{attribute 'linkalways'} 
{attribute 'no_explicit_call' := 'This FB is a CLASS and must be accessed using methods or properties'}
{attribute 'enable_dynamic_creation'}
FUNCTION_BLOCK PromiseContext IMPLEMENTS I_PromiseContext
VAR
	state : (PROMISE_PENDING, PROMISE_REJECTED, PROMISE_RESOLVED);
	reason : T_MAXSTRING;
	entities : Dictionary;
	pBuffer : POINTER TO BYTE;
	bufferSize : UDINT;
END_VAR

METHOD PRIVATE CopyBufferToDestination
VAR_INPUT
	DestinationAddress : PVOID;
END_VAR
MEMCPY(DestinationAddress, pBuffer, bufferSize);
END_METHOD

METHOD PRIVATE CopySourceToBuffer
VAR_INPUT
	SourceAddress : PVOID;
END_VAR
MEMCPY(pBuffer, SourceAddress, bufferSize);
END_METHOD

METHOD PRIVATE CreateBuffer
VAR_INPUT
	SizeInBytes : UDINT;
END_VAR
bufferSize := SizeInBytes;
pBuffer := __NEW(BYTE, SizeInBytes);
END_METHOD

METHOD PRIVATE DestroyBuffer
VAR_INPUT
END_VAR
IF pBuffer = 0 THEN
	RETURN;
END_IF

__DELETE(pBuffer);
bufferSize := 0;
END_METHOD

METHOD FB_exit : BOOL
VAR_INPUT
	bInCopyCode : BOOL; // if TRUE, the exit method is called for exiting an instance that is copied afterwards (online change).
END_VAR
IF bInCopyCode THEN
	RETURN;
END_IF

DestroyBuffer();
END_METHOD

PROPERTY PUBLIC Pending : BOOL
GET
Pending := state = PROMISE_PENDING;
END_GET
END_PROPERTY

METHOD PUBLIC Reject
VAR_INPUT
	Reason : T_MAXSTRING;
END_VAR
IF NOT Pending THEN
	RETURN;
END_IF

THIS^.reason := Reason;
state := PROMISE_REJECTED;
END_METHOD

PROPERTY Rejected : BOOL
GET
Rejected := state = PROMISE_REJECTED;
END_GET
END_PROPERTY

PROPERTY RejectedReason : T_MAXSTRING
GET
RejectedReason := reason;
END_GET
END_PROPERTY

METHOD PUBLIC Resolve
VAR_INPUT
END_VAR
IF NOT Pending THEN
	RETURN;
END_IF

state := PROMISE_RESOLVED;
END_METHOD

PROPERTY Resolved : BOOL
GET
Resolved := state = PROMISE_RESOLVED;
END_GET
END_PROPERTY

METHOD PUBLIC ResolveWith
VAR_INPUT
	Value : ANY;
END_VAR
IF NOT Pending THEN
	RETURN;
END_IF

state := PROMISE_RESOLVED;
CreateBuffer(DINT_TO_UDINT(Value.diSize));
CopySourceToBuffer(Value.pValue);
END_METHOD

METHOD PUBLIC TryGetEntity : BOOL
VAR_INPUT
	Key : T_MAXSTRING;
	Destination	: ANY;
END_VAR
TryGetEntity := entities.TryGetValue(Key, Destination);
END_METHOD

METHOD PUBLIC TryGetEntityTo : BOOL
VAR_INPUT
	Key : T_MAXSTRING;
	DestinationAddress : PVOID;
	DestinationSize : UDINT;
END_VAR
TryGetEntityTo := entities.TryGetValueTo(Key, DestinationAddress, DestinationSize);
END_METHOD

METHOD PUBLIC TryGetResult : BOOL
VAR_INPUT
	Destination : ANY;
END_VAR
IF NOT Resolved THEN
	RETURN;
END_IF

TryGetResult := TryGetResultTo(Destination.pValue, DINT_TO_UDINT(Destination.diSize));
END_METHOD

METHOD PUBLIC TryGetResultTo : BOOL
VAR_INPUT
	DestinationAddress : PVOID;
	DestinationSize : UDINT;
END_VAR
IF NOT Resolved THEN
	RETURN;
END_IF

IF pBuffer = 0 THEN
	RETURN;
END_IF

IF bufferSize <> DestinationSize THEN
	RETURN;
END_IF

CopyBufferToDestination(DestinationAddress);
TryGetResultTo := TRUE;
END_METHOD

METHOD PUBLIC TrySetEntity : BOOL
VAR_INPUT
	Key : T_MAXSTRING;
	Value : ANY;
END_VAR
TrySetEntity := entities.TryAdd(Key, Value);
END_METHOD

END_FUNCTION_BLOCK

(* stored: Version 1.1.0.1, ProductVersion 3.1.4024.12
   POU PromiseContext: Id {75de2a15-307e-435d-83d9-7a9c6fc0aa6b}, SpecialFunc None
   Folder Destructor: Id {3206c6d1-73ba-4bcb-9573-ef49dfe35813}
   Folder Private: Id {2aeb644b-aaad-4298-8cfb-e5854fe0a558}
   Method CopyBufferToDestination: Id {643053a8-761b-44b6-b0e6-941cdfc54020}
   Method CopySourceToBuffer: Id {18d0ddd0-a56f-44a7-8313-4f7aac18c40f}
   Method CreateBuffer: Id {d1c0e31e-bcae-46c4-a6b3-a9a2c7832b79}
   Method DestroyBuffer: Id {18a4e6b2-a240-42cc-907a-6394e5a913fc}
   Method FB_exit: Id {ed9e31bb-5056-4c6e-aecd-e284355dc15c}
   Property Pending: Id {3e6c5105-de16-4dc6-9419-c281f6072c9e}
   Get Get: Id {c8bcd943-4822-4043-8555-5d3c366f5060}
   Method Reject: Id {3005d554-6d2b-4118-bbde-742e87e3e26b}
   Property Rejected: Id {19b6e227-f6bc-4e54-bb57-3ef321fea3ee}
   Get Get: Id {a2e9ead9-bf2b-4df8-85d9-9300605aee90}
   Property RejectedReason: Id {54ee7955-fd3c-48fe-8732-72512e9a1ff9}
   Get Get: Id {f4b08042-2a5e-4864-8192-66c3e2b97f00}
   Method Resolve: Id {a6b23446-da8d-43df-9791-1e09c13c9a89}
   Property Resolved: Id {d82e39ea-5d83-4fc9-8332-fb4bab329fd2}
   Get Get: Id {f80a32f1-777d-40d0-807b-86ea3f5a0bc8}
   Method ResolveWith: Id {16016f5e-a90b-4a96-bfdf-2b6d1e39081f}
   Method TryGetEntity: Id {88900e9e-b119-4bf3-8c3f-0fad1d1aedb0}
   Method TryGetEntityTo: Id {24758a8f-073d-4e7a-92dc-9315e7ebb72c}
   Method TryGetResult: Id {cec1d925-83de-40ec-acf7-c0fa197cb481}
   Method TryGetResultTo: Id {ebc6e9b1-9d29-4747-b08d-763392ba9d46}
   Method TrySetEntity: Id {b791e364-d050-4f57-8a23-0d598e9a6c10} *)
